TEXTLIST TextList_Config_Gaz
  0 = 'gaz\t' | FR: 'Gaz' | EN: 'Gas'
  1 = 'definition gaz' | FR: 'Définition des gaz' | EN: 'Gas definition'
  2 = 'supervi gaz\t' | FR: 'Surveillance' | EN: 'Monitoring'
  3 = 'debit sccm' | FR: 'Tous les débits en sccm' | EN: 'All flows in sccm'
  4 = 'seuil sccm' | FR: 'Tous les seuils en sccm' | EN: 'All thresholds in sccm'
  5 = 'nom gaz nom' | FR: 'Nom du gaz\nnominal' | EN: 'Nominal\ngas name'
  6 = 'Coef' | FR: 'Coeff. de\nconversion' | EN: 'Conversion\ncoeff.'
  7 = 'debit max' | FR: 'Débit max.\ndébitmètre' | EN: 'Massflow\nmax. flow'
  8 = 'nom gaz util' | FR: 'Nom du gaz\nutilisé' | EN: 'Used gas\nname'
  9 = 'debi max gaz' | FR: 'Débit max.\ngaz' | EN: 'Gas\nmax. flow'
  11 = 'gaz1' | FR: 'Gaz 1' | EN: 'Gas 1'
  12 = 'gaz 2' | FR: 'Gaz 2' | EN: 'Gas 2'
  13 = 'gaz 3' | FR: 'Gaz 3' | EN: 'Gas 3'
  14 = 'gaz 4' | FR: 'Gaz 4' | EN: 'Gas 4'
  15 = 'gaz 5' | FR: 'Gaz 5' | EN: 'Gas 5'
  16 = 'gaz 6' | FR: 'Gaz 6' | EN: 'Gas 6'
  17 = 'gaz7' | FR: 'Gaz 7' | EN: 'Gas 7'
  18 = 'gaz8' | FR: 'Gaz 8' | EN: 'Gas 8'
  19 = 'gaz9' | FR: 'Gaz 9' | EN: 'Gas 9'
  20 = 'seuil alarme' | FR: "Seuil\nd'alarme" | EN: 'Alarm\nthreshold'
  21 = 'tps alarm' | FR: 'Temps avant\nalarme' | EN: 'Alarm\ndelay'
  22 = 'seuil défaut' | FR: 'Seuil\nde défaut' | EN: 'Fault\nthreshold'
  23 = 'tps défaut' | FR: 'Temps avant\ndéfaut' | EN: 'Fault\ndelay'
  10 = 'Purge canon' | FR: 'Purge canons à ions' | EN: 'Ions beam purge'
  24 = "Purge d'amo" | FR: "Purge d'amorcage" | EN: 'Start purge'
  25 = 'Purge stop' | FR: "Purge d'arrêt" | EN: 'Purge stop'
  26 = 'Durée' | FR: 'Durée' | EN: 'Duration'
  27 = 'Purge RAH' | FR: 'Purge atmosphère' | EN: 'Atmospheric purge'
  28 = 'Rapide' | FR: 'Rapide' | EN: 'Fast'
  29 = 'Ala surv press' | FR: 'Surveillance pression - Temps avant alarme' | EN: 'Pressure supervision - Delay before alarm'
  30 = 'def surv press' | FR: 'Surveillance pression - Temps avant défaut' | EN: 'Pressure supervision - Delay before default'
  31 = 'Gain' | FR: 'Gain' | EN: 'Amplification factor'
  32 = 'Ti' | FR: "Temps d'action intégrale" | EN: 'Integral action time'
  33 = 'Td' | FR: "Temps d'action dérivée" | EN: 'Derivative action time '
  34 = 'Ta' | FR: "Temps d'amortissment" | EN: 'Damping time'
  35 = 'Regul Gaz' | FR: 'Régulation de gaz' | EN: 'Gas regulation'
   = ''
END_TEXTLIST

(* stored: Version 1.1.0.1, ProductVersion 3.1.4024.10
   TextList TextList_Config_Gaz: Id {d999b0cd-6657-417a-89eb-35c59fa7a078} *)
